(* Logix 5000 project; controller NSH_PLC1 vendor 1 type 14 code 167 rev 32.11; software revision 32.02; part 10 of 12 *)
(* tags used below, declared in another part *)
   BH3 : Motor;   // BH Rock
   CR_RunCommon : BOOL;   // PreClean, Run Common Units
   CR_StopCommon : BOOL;   // PreClean, Stop Common Units
   CR_StopLine1 : BOOL;   // Pre Clean Stop Line 1 Relay
   CR_StopPC1_FansCO : BOOL;   // Pre Clean Stop Line 1 Fans Cleanout Relay
   CR_StopPC2_FansCO : BOOL;   // Pre Clean Stop Line 2 Fans Cleanout Relay
   DummyOutput : BOOL;
   MainBin1 : MainBins;   // PreClean to Huller, Main Bin #1
   MainBin2 : MainBins;   // PreClean to Huller, Main Bin #1
   MainBin3 : MainBins;   // PreClean to Huller, Main Bin #1
   MainBin4 : MainBins;   // PreClean to Huller, Main Bin #1
   MainBin5 : MainBins;   // PreClean to Huller, Main Bin #1
   MainBin6 : MainBins;   // PreClean to Huller, Main Bin #1
   MainBin7 : MainBins;   // PreClean to Huller, Main Bin #1
   MainBin8 : MainBins;   // PreClean to Huller, Main Bin #1
   P10_5A : Motor;   // Cross Auger
   P10A : Motor;   // Elev to Bins
   P11A : Motor;   // Line1 Auger
   P11B : Motor;   // Line2 Auger
   P1A : Motor;   // DO Conv.
   P2A : Motor;   // Cross Conv.
   P3A : Motor;   // Stick Reel
   P4A : Motor;   // C. Belt
   P5A : Motor;   // Ele. to Vib
   P6A : Motor;   // Vib Splitter
   P7A : Motor;   // Screener
   P7A1 : Motor;   // Screener
   P7A2 : Motor;   // Screener
   P8A2_A : Motor;   // Destoner
   P8A2_B : Motor;   // AirLock
   P8A_A : Motor;   // Destoner
   P8A_B : Motor;   // Airlock
   P9A : Motor;   // Auger
   PBB1A : Motor;   // AirLock
   PBB2A : Motor;   // AirLock
   PD1 : Motor;   // Dirt Conv.
   PD2 : Motor;   // Incline
   PR1 : Motor;   // Rock Conv.
   PR2 : Motor;   // Inc. Rock
   PR3 : Motor;   // Belt
   PS1 : Motor;   // Stick Conv.
   PS2 : Motor;   // Inc. Stick Conv.
   PS3 : Motor;   // Twig Conv.
   PS4 : Motor;   // Twig Conv.
   TMR_LineStart1 : TIMER;   // Pre Clean Line 1 Start Warning Timer
   TMR_LineStart2 : TIMER;   // Pre Clean Line 2 Start Warning Timer
   TMR_StartPC1_FansCO : TIMER;   // Pre Clean Line 1 Fans Cleanout Start Warning Timer
   TMR_StartPC2_FansCO : TIMER;   // Pre Clean Line 2 Fans Cleanout Start Warning Timer
(* MainProgram, continued *)

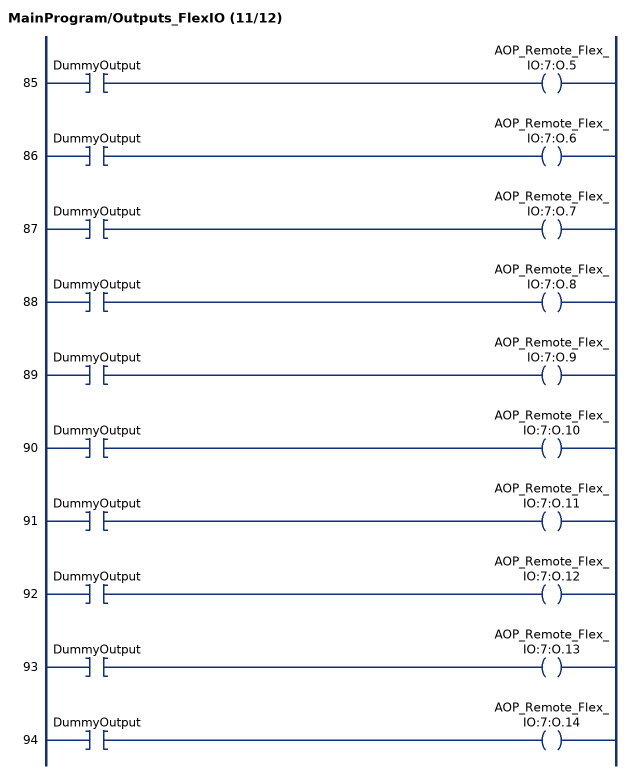
   [picture p210: MainProgram/Outputs_FlexIO rungs 85-94]
   85: XIC(DummyOutput)OTE(AOP_Remote_Flex_IO:7:O.5);
   86: XIC(DummyOutput)OTE(AOP_Remote_Flex_IO:7:O.6);
   87: XIC(DummyOutput)OTE(AOP_Remote_Flex_IO:7:O.7);
   88: XIC(DummyOutput)OTE(AOP_Remote_Flex_IO:7:O.8);
   89: XIC(DummyOutput)OTE(AOP_Remote_Flex_IO:7:O.9);
   90: XIC(DummyOutput)OTE(AOP_Remote_Flex_IO:7:O.10);
   91: XIC(DummyOutput)OTE(AOP_Remote_Flex_IO:7:O.11);
   92: XIC(DummyOutput)OTE(AOP_Remote_Flex_IO:7:O.12);
   93: XIC(DummyOutput)OTE(AOP_Remote_Flex_IO:7:O.13);
   94: XIC(DummyOutput)OTE(AOP_Remote_Flex_IO:7:O.14);
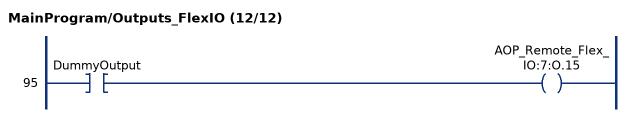
   95: XIC(DummyOutput)OTE(AOP_Remote_Flex_IO:7:O.15);
END_ROUTINE

ROUTINE Outputs_MCC1   (* ladder *)
END_ROUTINE

ROUTINE Outputs_PLC2_MCC2   (* ladder *)
END_ROUTINE

ROUTINE Outputs_PLC2_MCC3   (* ladder *)
END_ROUTINE

ROUTINE PF525_AOP_ToMotorsSUB   (* ladder *)
// Get PowerFlex525 AOP Inputs and Put Into Motor Structure
END_ROUTINE

ROUTINE PF755_AOP_ToMotorsSUB   (* ladder *)
// Get PowerFlex755 AOP Inputs and Put Into Motor Structure
END_ROUTINE
END_PROGRAM

PROGRAM PreClean   (* main routine PC_MainJSR *)
// PreClean
VAR
   CTR_HornBeeps : COUNTER := (PRE := 3);   // Number of times horn beeps
   FaultPresent : BOOL;   // A PreClean Fault is Present
   FaultReset : BOOL;   // PreClean Fault Reset
   NewFault : BOOL;   // New Precelan Fault has just occured
   NewFaultBeepHorn : BOOL;   // New Alarm, Pulse Horn
   Num_Faults : DINT;   // Number of PreCelan Faults
   Num_Faults_LS : DINT;   // Number of PreCelan Faults Last PLC Scan
   Num_Warnings : DINT;   // Number of PreCelan Warnings
   Reset_TOF_PRE : DINT;   // Reset pulse duration to Drives
   SpeedIsFactored : BOOL;   // Speed of VFD is factored by Master Speed Factor
   TempAccelerating : BOOL;   // Temp Motor is Accelerating
   TempActive : BOOL;   // Temp Motor is Active
   TempAlarm : BOOL;   // Temp Motor has Alarm
   TempAtSpeed : BOOL;   // Temp Motor is At Speed
   TempCommAlarm : BOOL;   // Temp Motor, AOP communications Alarm
   TempDecelerating : BOOL;   // Temp Motor is Decelerating
   TempFaulted : BOOL;   // Temp Motor is Faulted
   TempImbalanceTrip : BOOL;   // Temp Motor, Phase Imbalance Trip
   TempImbalanceWarning : BOOL;   // Temp Motor, Phase Imbalance Warning
   TempMainBin : MainBins := (TMR_BinFull.PRE := 20000, TMR_BinNotFull.PRE := 20000);   // Main Bin Temp
   TempMotor : Motor := (Fault_TON.PRE := 1000, Warning_TON.PRE := 1000, Reset_TOF.PRE := 500); {access None}
   TempOL_Percent : DINT;   // Temp Motor Percent Overload
   TempOverloadTrip : BOOL;   // Temp Motor, Overload Trip
   TempOverloadWarning : BOOL;   // Temp Motor, Overlaod Warning
   TempPhaseLossTrip : BOOL;   // Temp Motor, Phase Loss Trip
   TempReady : BOOL;   // Temp Motor is ready
   TempRunning : BOOL;   // Temp Motor is Running
   TempTriped : BOOL;   // Temp Motor Tripped
   TempVFD : VFD_Extra;   // Temp VFD Structure
   TempWarning : BOOL;   // Temp Motor Warning
   TMR_HornFlasher : TIMER := (PRE := 1000);   // Fault Horn Flasher timer
END_VAR

ROUTINE E300_StatusAlmWarnSUB   (* ladder *)
// Decode Status Bits and Set Warnings and Alarms For NRFV Motors with E300
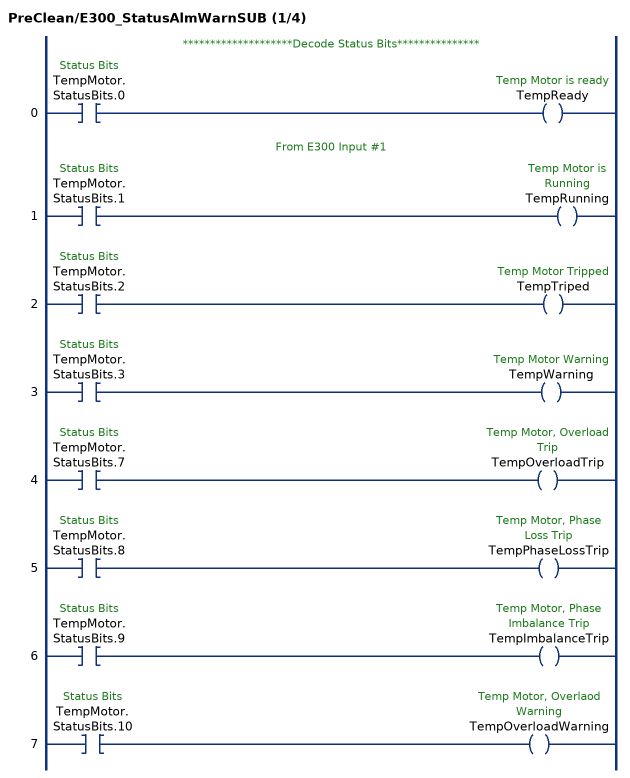
   // ********************Decode Status Bits***************
   0: XIC(TempMotor.StatusBits.0)OTE(TempReady);
   // From E300 Input #1
   1: XIC(TempMotor.StatusBits.1)OTE(TempRunning);
   2: XIC(TempMotor.StatusBits.2)OTE(TempTriped);
   3: XIC(TempMotor.StatusBits.3)OTE(TempWarning);
   4: XIC(TempMotor.StatusBits.7)OTE(TempOverloadTrip);
   5: XIC(TempMotor.StatusBits.8)OTE(TempPhaseLossTrip);
   6: XIC(TempMotor.StatusBits.9)OTE(TempImbalanceTrip);
   7: XIC(TempMotor.StatusBits.10)OTE(TempOverloadWarning);
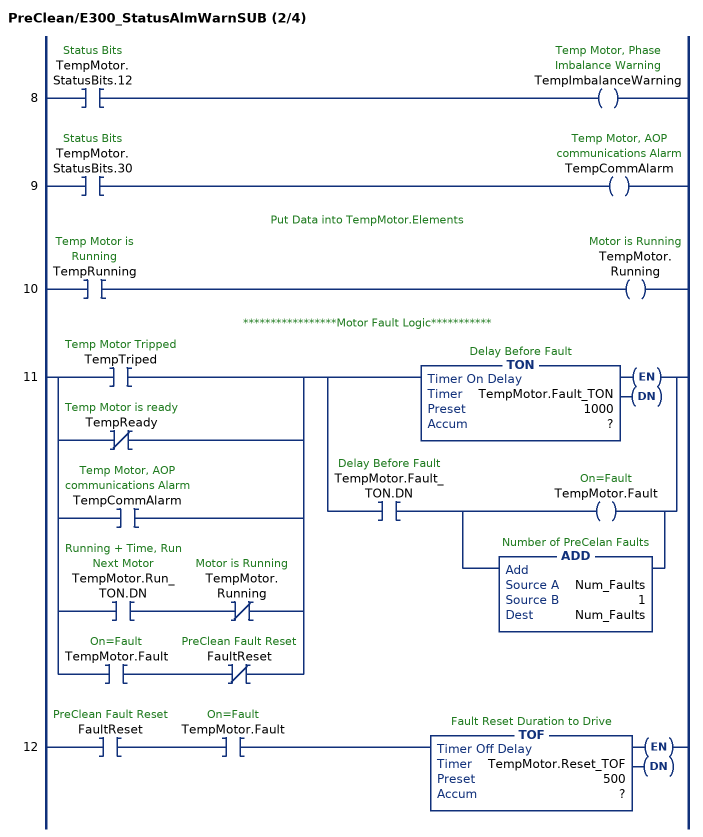
   8: XIC(TempMotor.StatusBits.12)OTE(TempImbalanceWarning);
   9: XIC(TempMotor.StatusBits.30)OTE(TempCommAlarm);
   // Put Data into TempMotor.Elements
   10: XIC(TempRunning)OTE(TempMotor.Running);
   // *****************Motor Fault Logic***********
   11: [XIC(TempTriped) ,XIO(TempReady) ,XIC(TempCommAlarm) ,XIC(TempMotor.Run_TON.DN) XIO(TempMotor.Running) ,XIC(TempMotor.Fault) XIO(FaultReset) ][TON(TempMotor.Fault_TON,?,?) ,XIC(TempMotor.Fault_TON.DN) [OTE(TempMotor.Fault) ,ADD(Num_Faults,1,Num_Faults) ] ];
   12: XIC(FaultReset)XIC(TempMotor.Fault)TOF(TempMotor.Reset_TOF,?,?);
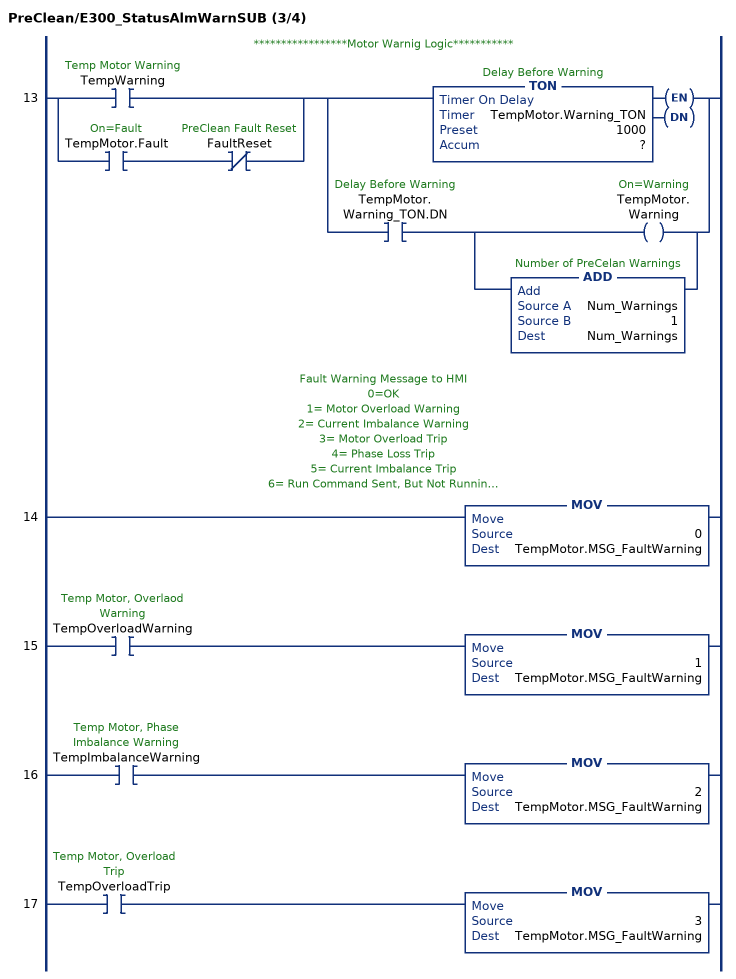
   // *****************Motor Warnig Logic***********
   13: [XIC(TempWarning) ,XIC(TempMotor.Fault) XIO(FaultReset) ][TON(TempMotor.Warning_TON,?,?) ,XIC(TempMotor.Warning_TON.DN) [OTE(TempMotor.Warning) ,ADD(Num_Warnings,1,Num_Warnings) ] ];
   // Fault Warning Message to HMI
   // 0=OK
   // 1= Motor Overload Warning
   // 2= Current Imbalance Warning
   // 3= Motor Overload Trip
   // 4= Phase Loss Trip
   // 5= Current Imbalance Trip
   // 6= Run Command Sent, But Not Running
   // 7=Loss Of Ethernet Communications
   // 8=VFD Fault
   14: MOV(0,TempMotor.MSG_FaultWarning);
   15: XIC(TempOverloadWarning)MOV(1,TempMotor.MSG_FaultWarning);
   16: XIC(TempImbalanceWarning)MOV(2,TempMotor.MSG_FaultWarning);
   17: XIC(TempOverloadTrip)MOV(3,TempMotor.MSG_FaultWarning);
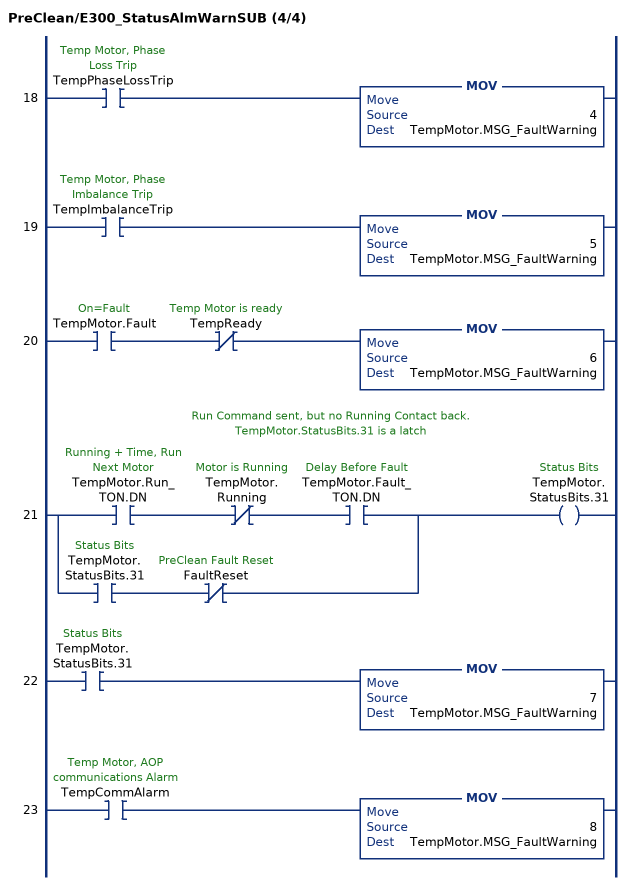
   18: XIC(TempPhaseLossTrip)MOV(4,TempMotor.MSG_FaultWarning);
   19: XIC(TempImbalanceTrip)MOV(5,TempMotor.MSG_FaultWarning);
   20: XIC(TempMotor.Fault)XIO(TempReady)MOV(6,TempMotor.MSG_FaultWarning);
   // Run Command sent, but no Running Contact back.
   // TempMotor.StatusBits.31 is a latch
   21: [XIC(TempMotor.Run_TON.DN) XIO(TempMotor.Running) XIC(TempMotor.Fault_TON.DN) ,XIC(TempMotor.StatusBits.31) XIO(FaultReset) ]OTE(TempMotor.StatusBits.31);
   22: XIC(TempMotor.StatusBits.31)MOV(7,TempMotor.MSG_FaultWarning);
   23: XIC(TempCommAlarm)MOV(8,TempMotor.MSG_FaultWarning);
END_ROUTINE

ROUTINE MainBins   (* ladder *)
// Control Main Bins
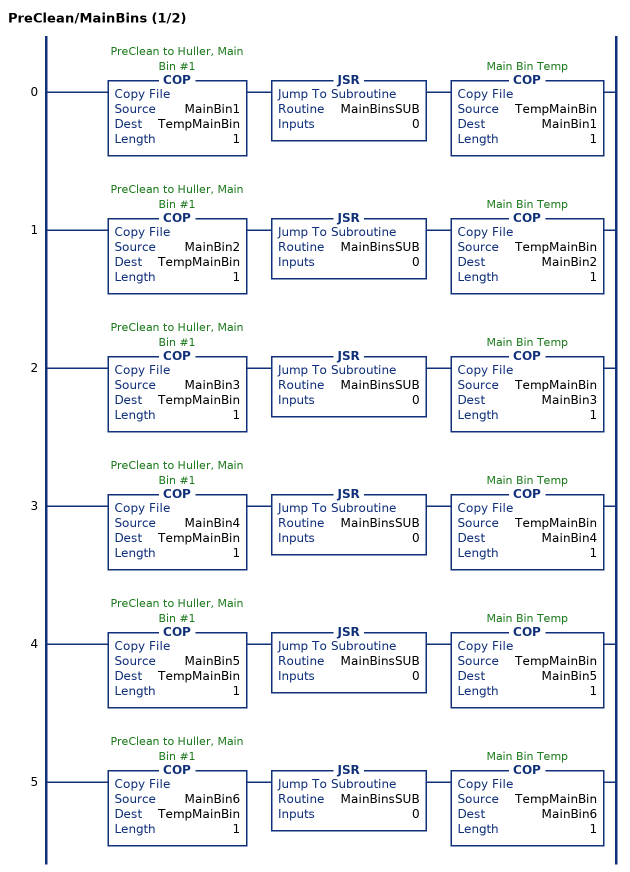
   0: COP(MainBin1,TempMainBin,1)JSR(MainBinsSUB,0)COP(TempMainBin,MainBin1,1);
   1: COP(MainBin2,TempMainBin,1)JSR(MainBinsSUB,0)COP(TempMainBin,MainBin2,1);
   2: COP(MainBin3,TempMainBin,1)JSR(MainBinsSUB,0)COP(TempMainBin,MainBin3,1);
   3: COP(MainBin4,TempMainBin,1)JSR(MainBinsSUB,0)COP(TempMainBin,MainBin4,1);
   4: COP(MainBin5,TempMainBin,1)JSR(MainBinsSUB,0)COP(TempMainBin,MainBin5,1);
   5: COP(MainBin6,TempMainBin,1)JSR(MainBinsSUB,0)COP(TempMainBin,MainBin6,1);
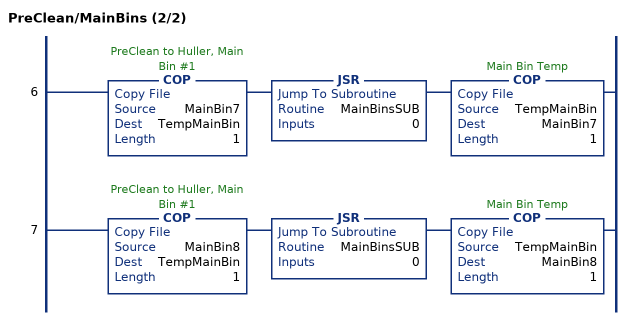
   6: COP(MainBin7,TempMainBin,1)JSR(MainBinsSUB,0)COP(TempMainBin,MainBin7,1);
   7: COP(MainBin8,TempMainBin,1)JSR(MainBinsSUB,0)COP(TempMainBin,MainBin8,1);
END_ROUTINE

ROUTINE MainBinsSUB   (* ladder *)
// Control Main Bins Switches and Lights
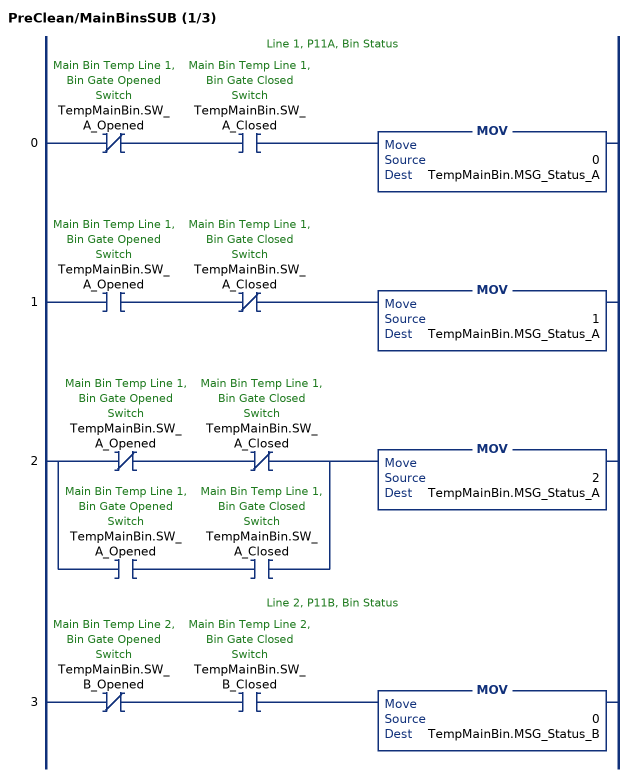
   // Line 1, P11A, Bin Status
   0: XIO(TempMainBin.SW_A_Opened)XIC(TempMainBin.SW_A_Closed)MOV(0,TempMainBin.MSG_Status_A);
   1: XIC(TempMainBin.SW_A_Opened)XIO(TempMainBin.SW_A_Closed)MOV(1,TempMainBin.MSG_Status_A);
   2: [XIO(TempMainBin.SW_A_Opened) XIO(TempMainBin.SW_A_Closed) ,XIC(TempMainBin.SW_A_Opened) XIC(TempMainBin.SW_A_Closed) ]MOV(2,TempMainBin.MSG_Status_A);
   // Line 2, P11B, Bin Status
   3: XIO(TempMainBin.SW_B_Opened)XIC(TempMainBin.SW_B_Closed)MOV(0,TempMainBin.MSG_Status_B);
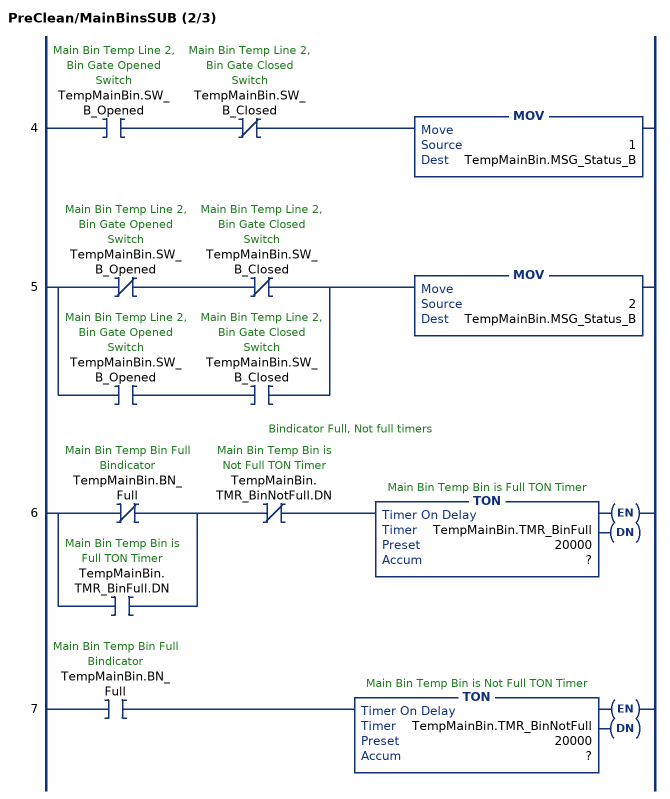
   4: XIC(TempMainBin.SW_B_Opened)XIO(TempMainBin.SW_B_Closed)MOV(1,TempMainBin.MSG_Status_B);
   5: [XIO(TempMainBin.SW_B_Opened) XIO(TempMainBin.SW_B_Closed) ,XIC(TempMainBin.SW_B_Opened) XIC(TempMainBin.SW_B_Closed) ]MOV(2,TempMainBin.MSG_Status_B);
   // Bindicator Full, Not full timers
   6: [XIO(TempMainBin.BN_Full) ,XIC(TempMainBin.TMR_BinFull.DN) ]XIO(TempMainBin.TMR_BinNotFull.DN)TON(TempMainBin.TMR_BinFull,?,?);
   7: XIC(TempMainBin.BN_Full)TON(TempMainBin.TMR_BinNotFull,?,?);
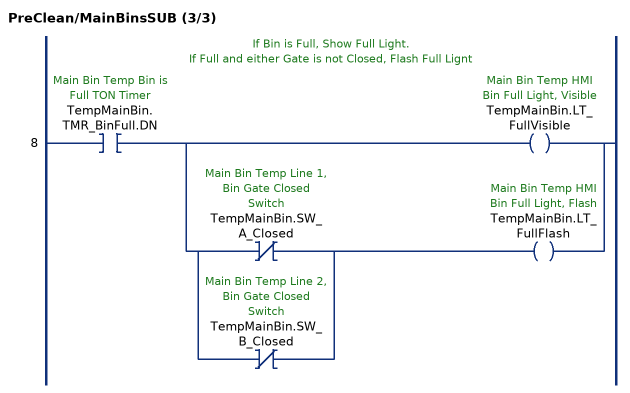
   // If Bin is Full, Show Full Light.
   // If Full and either Gate is not Closed, Flash Full Lignt
   8: XIC(TempMainBin.TMR_BinFull.DN)[OTE(TempMainBin.LT_FullVisible) ,[XIO(TempMainBin.SW_A_Closed) ,XIO(TempMainBin.SW_B_Closed) ] OTE(TempMainBin.LT_FullFlash) ];
END_ROUTINE

ROUTINE Motors   (* ladder *)
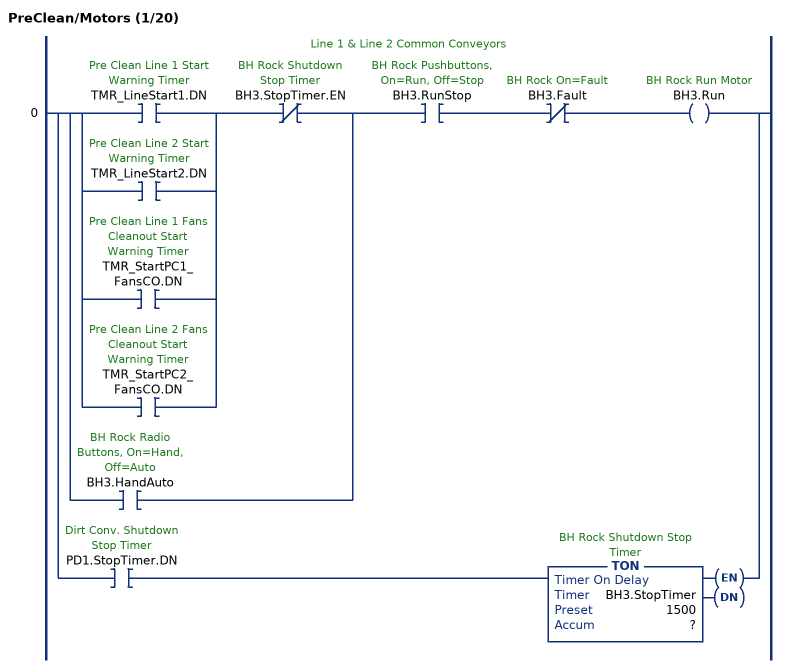
   // Line 1 & Line 2 Common Conveyors
   0: [[[XIC(TMR_LineStart1.DN) ,XIC(TMR_LineStart2.DN) ,XIC(TMR_StartPC1_FansCO.DN) ,XIC(TMR_StartPC2_FansCO.DN) ] XIO(BH3.StopTimer.EN) ,XIC(BH3.HandAuto) ] XIC(BH3.RunStop) XIO(BH3.Fault) OTE(BH3.Run) ,XIC(PD1.StopTimer.DN) TON(BH3.StopTimer,?,?) ];
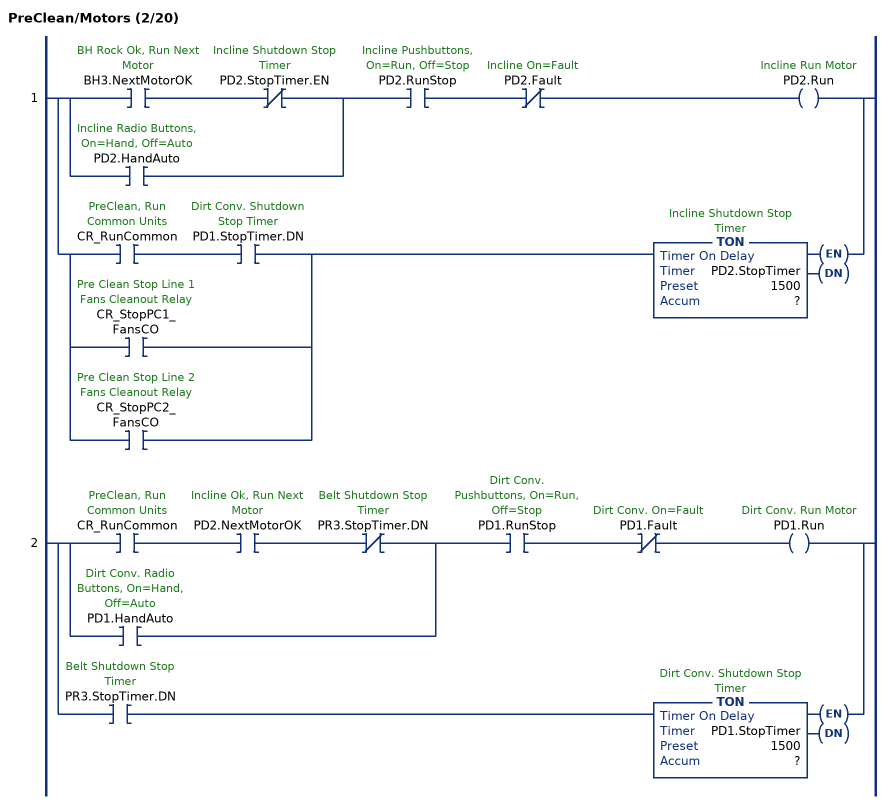
   1: [[XIC(BH3.NextMotorOK) XIO(PD2.StopTimer.EN) ,XIC(PD2.HandAuto) ] XIC(PD2.RunStop) XIO(PD2.Fault) OTE(PD2.Run) ,[XIC(CR_RunCommon) XIC(PD1.StopTimer.DN) ,XIC(CR_StopPC1_FansCO) ,XIC(CR_StopPC2_FansCO) ] TON(PD2.StopTimer,?,?) ];
   2: [[XIC(CR_RunCommon) XIC(PD2.NextMotorOK) XIO(PR3.StopTimer.DN) ,XIC(PD1.HandAuto) ] XIC(PD1.RunStop) XIO(PD1.Fault) OTE(PD1.Run) ,XIC(PR3.StopTimer.DN) TON(PD1.StopTimer,?,?) ];
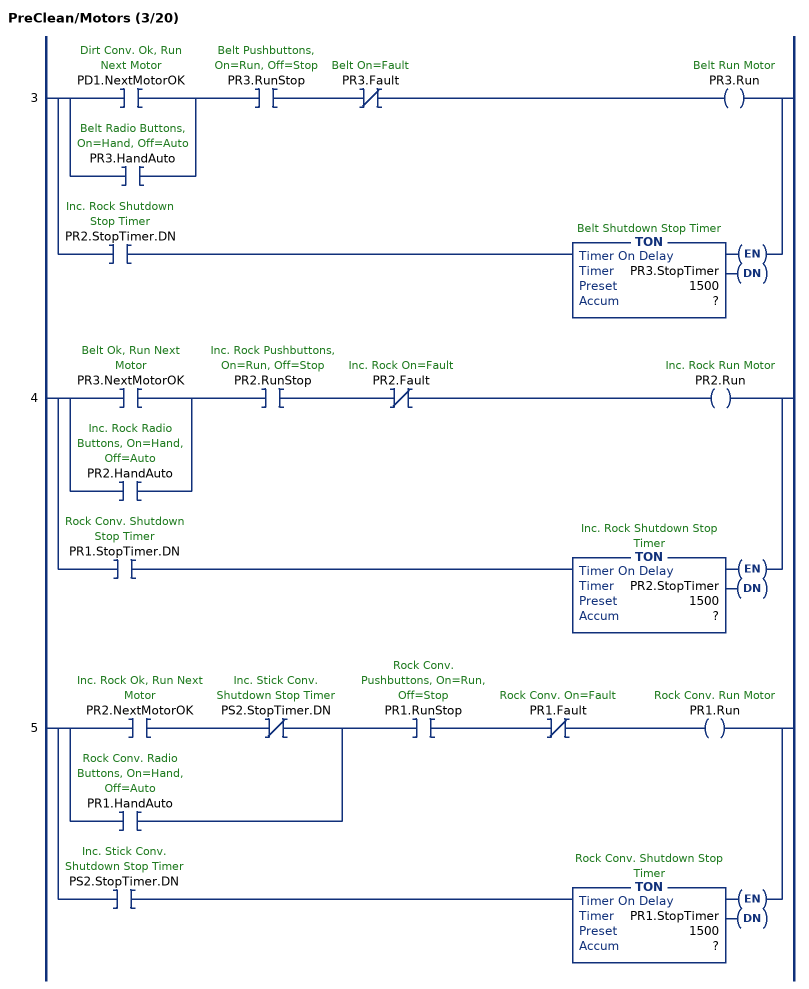
   3: [[XIC(PD1.NextMotorOK) ,XIC(PR3.HandAuto) ] XIC(PR3.RunStop) XIO(PR3.Fault) OTE(PR3.Run) ,XIC(PR2.StopTimer.DN) TON(PR3.StopTimer,?,?) ];
   4: [[XIC(PR3.NextMotorOK) ,XIC(PR2.HandAuto) ] XIC(PR2.RunStop) XIO(PR2.Fault) OTE(PR2.Run) ,XIC(PR1.StopTimer.DN) TON(PR2.StopTimer,?,?) ];
   5: [[XIC(PR2.NextMotorOK) XIO(PS2.StopTimer.DN) ,XIC(PR1.HandAuto) ] XIC(PR1.RunStop) XIO(PR1.Fault) OTE(PR1.Run) ,XIC(PS2.StopTimer.DN) TON(PR1.StopTimer,?,?) ];
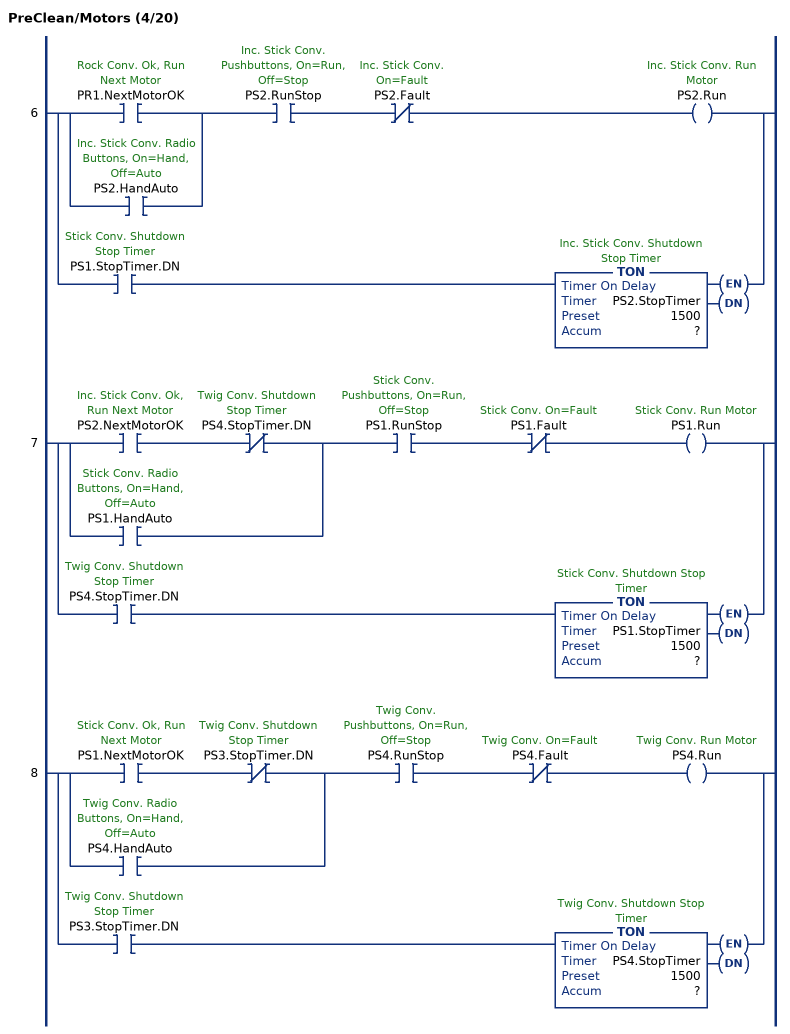
   6: [[XIC(PR1.NextMotorOK) ,XIC(PS2.HandAuto) ] XIC(PS2.RunStop) XIO(PS2.Fault) OTE(PS2.Run) ,XIC(PS1.StopTimer.DN) TON(PS2.StopTimer,?,?) ];
   7: [[XIC(PS2.NextMotorOK) XIO(PS4.StopTimer.DN) ,XIC(PS1.HandAuto) ] XIC(PS1.RunStop) XIO(PS1.Fault) OTE(PS1.Run) ,XIC(PS4.StopTimer.DN) TON(PS1.StopTimer,?,?) ];
   8: [[XIC(PS1.NextMotorOK) XIO(PS3.StopTimer.DN) ,XIC(PS4.HandAuto) ] XIC(PS4.RunStop) XIO(PS4.Fault) OTE(PS4.Run) ,XIC(PS3.StopTimer.DN) TON(PS4.StopTimer,?,?) ];
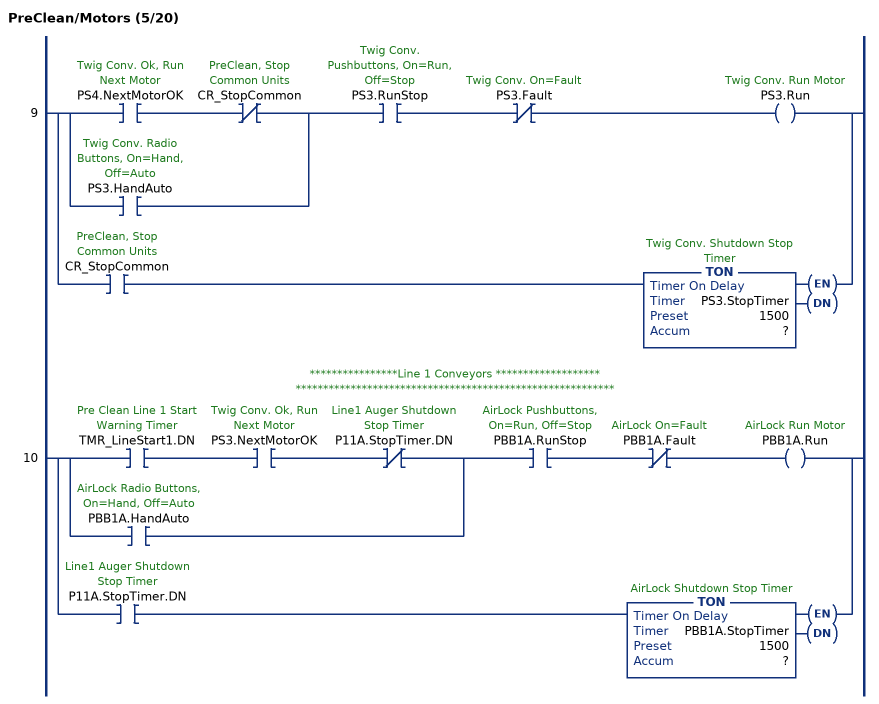
   9: [[XIC(PS4.NextMotorOK) XIO(CR_StopCommon) ,XIC(PS3.HandAuto) ] XIC(PS3.RunStop) XIO(PS3.Fault) OTE(PS3.Run) ,XIC(CR_StopCommon) TON(PS3.StopTimer,?,?) ];
   // ****************Line 1 Conveyors *******************
   //  **********************************************************
   10: [[XIC(TMR_LineStart1.DN) XIC(PS3.NextMotorOK) XIO(P11A.StopTimer.DN) ,XIC(PBB1A.HandAuto) ] XIC(PBB1A.RunStop) XIO(PBB1A.Fault) OTE(PBB1A.Run) ,XIC(P11A.StopTimer.DN) TON(PBB1A.StopTimer,?,?) ];
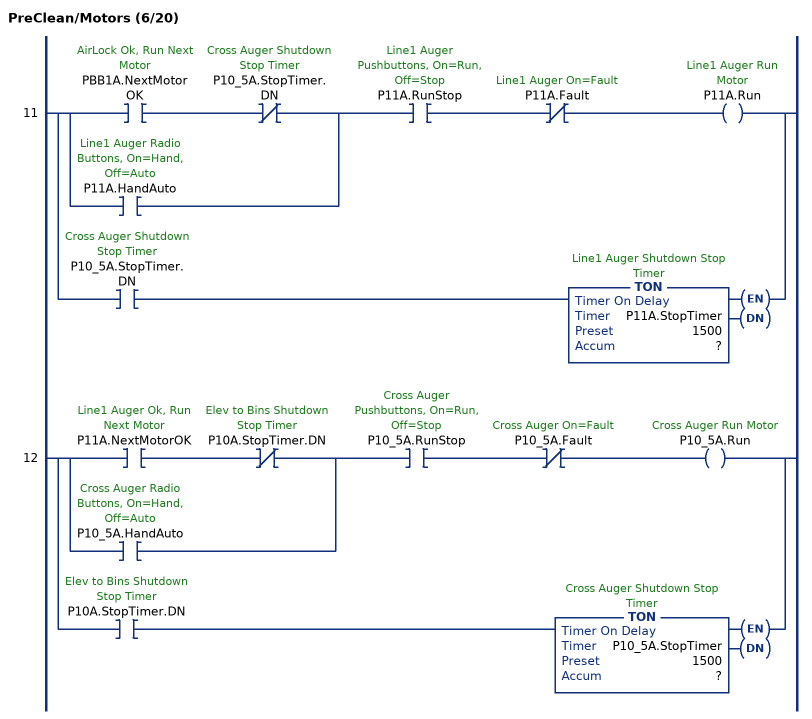
   11: [[XIC(PBB1A.NextMotorOK) XIO(P10_5A.StopTimer.DN) ,XIC(P11A.HandAuto) ] XIC(P11A.RunStop) XIO(P11A.Fault) OTE(P11A.Run) ,XIC(P10_5A.StopTimer.DN) TON(P11A.StopTimer,?,?) ];
   12: [[XIC(P11A.NextMotorOK) XIO(P10A.StopTimer.DN) ,XIC(P10_5A.HandAuto) ] XIC(P10_5A.RunStop) XIO(P10_5A.Fault) OTE(P10_5A.Run) ,XIC(P10A.StopTimer.DN) TON(P10_5A.StopTimer,?,?) ];
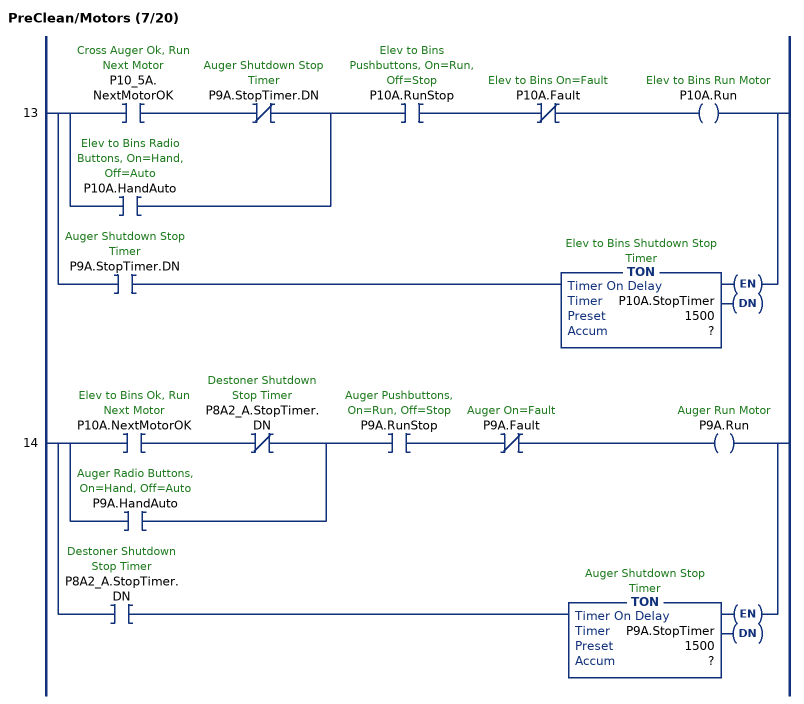
   13: [[XIC(P10_5A.NextMotorOK) XIO(P9A.StopTimer.DN) ,XIC(P10A.HandAuto) ] XIC(P10A.RunStop) XIO(P10A.Fault) OTE(P10A.Run) ,XIC(P9A.StopTimer.DN) TON(P10A.StopTimer,?,?) ];
   14: [[XIC(P10A.NextMotorOK) XIO(P8A2_A.StopTimer.DN) ,XIC(P9A.HandAuto) ] XIC(P9A.RunStop) XIO(P9A.Fault) OTE(P9A.Run) ,XIC(P8A2_A.StopTimer.DN) TON(P9A.StopTimer,?,?) ];
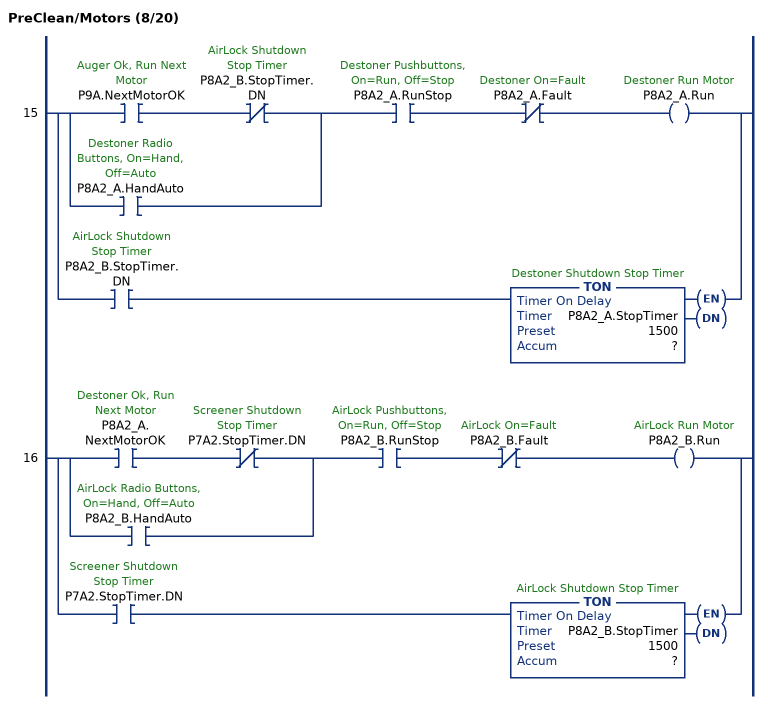
   15: [[XIC(P9A.NextMotorOK) XIO(P8A2_B.StopTimer.DN) ,XIC(P8A2_A.HandAuto) ] XIC(P8A2_A.RunStop) XIO(P8A2_A.Fault) OTE(P8A2_A.Run) ,XIC(P8A2_B.StopTimer.DN) TON(P8A2_A.StopTimer,?,?) ];
   16: [[XIC(P8A2_A.NextMotorOK) XIO(P7A2.StopTimer.DN) ,XIC(P8A2_B.HandAuto) ] XIC(P8A2_B.RunStop) XIO(P8A2_B.Fault) OTE(P8A2_B.Run) ,XIC(P7A2.StopTimer.DN) TON(P8A2_B.StopTimer,?,?) ];
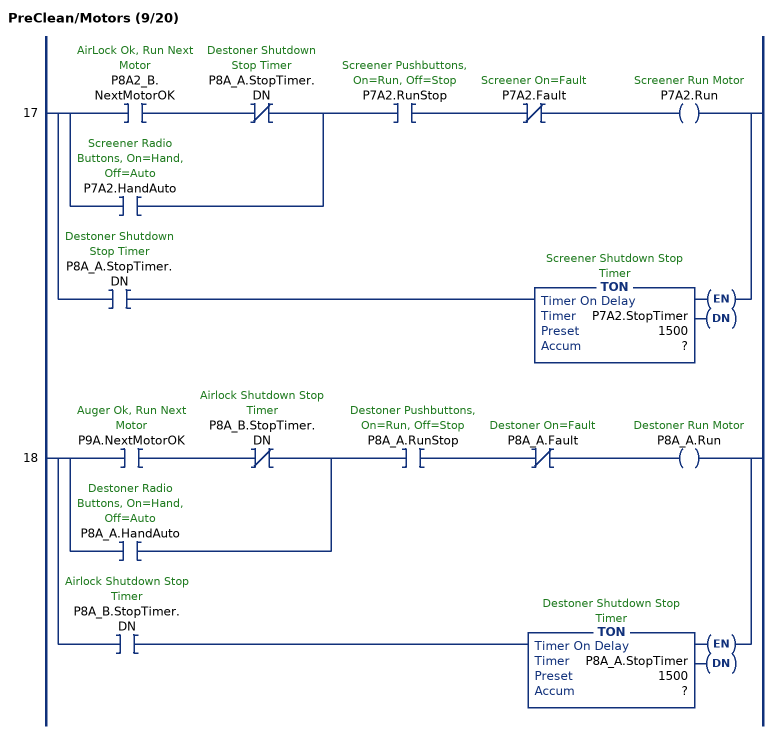
   17: [[XIC(P8A2_B.NextMotorOK) XIO(P8A_A.StopTimer.DN) ,XIC(P7A2.HandAuto) ] XIC(P7A2.RunStop) XIO(P7A2.Fault) OTE(P7A2.Run) ,XIC(P8A_A.StopTimer.DN) TON(P7A2.StopTimer,?,?) ];
   18: [[XIC(P9A.NextMotorOK) XIO(P8A_B.StopTimer.DN) ,XIC(P8A_A.HandAuto) ] XIC(P8A_A.RunStop) XIO(P8A_A.Fault) OTE(P8A_A.Run) ,XIC(P8A_B.StopTimer.DN) TON(P8A_A.StopTimer,?,?) ];
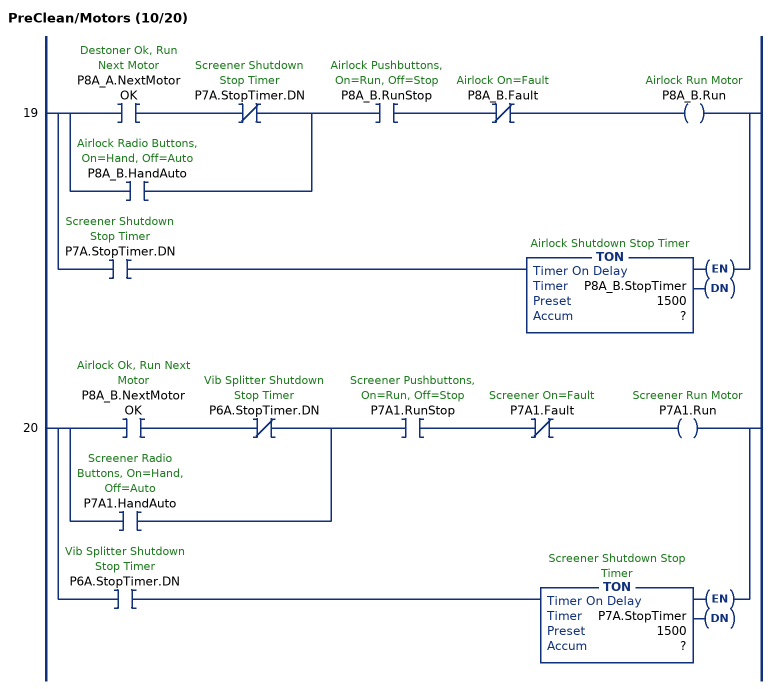
   19: [[XIC(P8A_A.NextMotorOK) XIO(P7A.StopTimer.DN) ,XIC(P8A_B.HandAuto) ] XIC(P8A_B.RunStop) XIO(P8A_B.Fault) OTE(P8A_B.Run) ,XIC(P7A.StopTimer.DN) TON(P8A_B.StopTimer,?,?) ];
   20: [[XIC(P8A_B.NextMotorOK) XIO(P6A.StopTimer.DN) ,XIC(P7A1.HandAuto) ] XIC(P7A1.RunStop) XIO(P7A1.Fault) OTE(P7A1.Run) ,XIC(P6A.StopTimer.DN) TON(P7A.StopTimer,?,?) ];
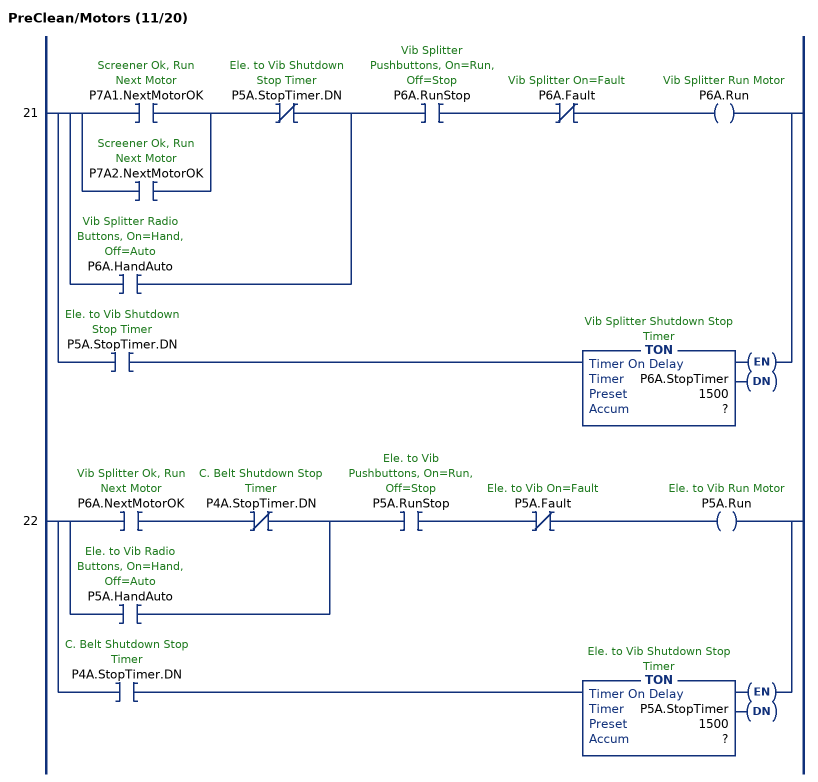
   21: [[[XIC(P7A1.NextMotorOK) ,XIC(P7A2.NextMotorOK) ] XIO(P5A.StopTimer.DN) ,XIC(P6A.HandAuto) ] XIC(P6A.RunStop) XIO(P6A.Fault) OTE(P6A.Run) ,XIC(P5A.StopTimer.DN) TON(P6A.StopTimer,?,?) ];
   22: [[XIC(P6A.NextMotorOK) XIO(P4A.StopTimer.DN) ,XIC(P5A.HandAuto) ] XIC(P5A.RunStop) XIO(P5A.Fault) OTE(P5A.Run) ,XIC(P4A.StopTimer.DN) TON(P5A.StopTimer,?,?) ];
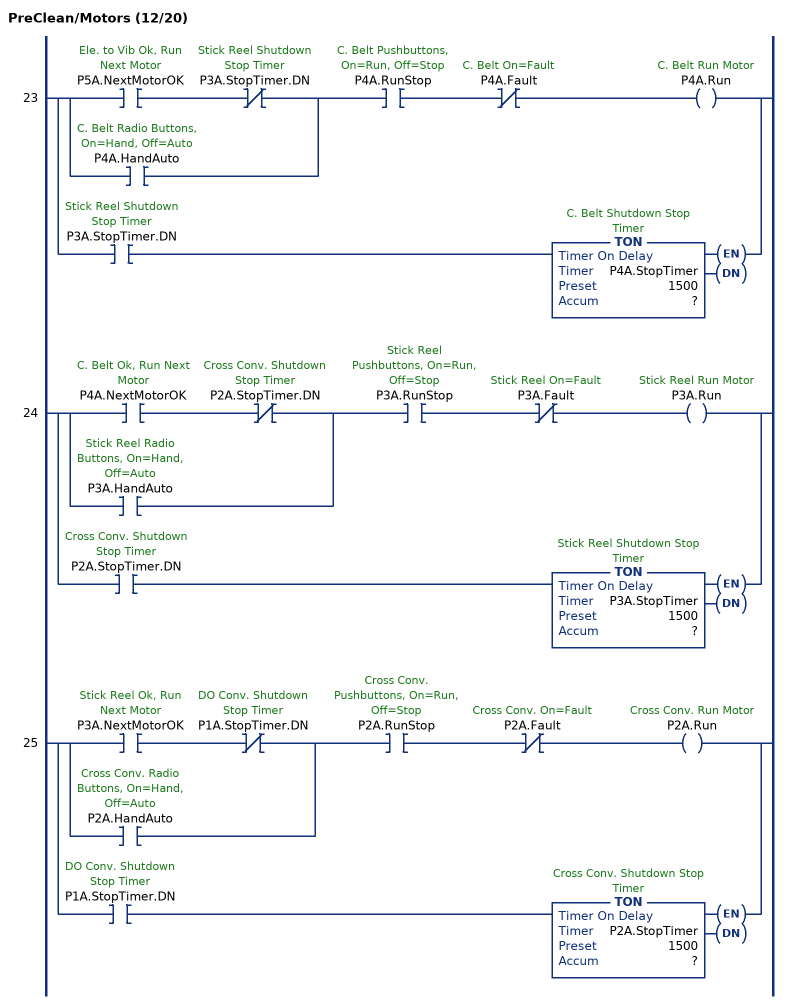
   23: [[XIC(P5A.NextMotorOK) XIO(P3A.StopTimer.DN) ,XIC(P4A.HandAuto) ] XIC(P4A.RunStop) XIO(P4A.Fault) OTE(P4A.Run) ,XIC(P3A.StopTimer.DN) TON(P4A.StopTimer,?,?) ];
   24: [[XIC(P4A.NextMotorOK) XIO(P2A.StopTimer.DN) ,XIC(P3A.HandAuto) ] XIC(P3A.RunStop) XIO(P3A.Fault) OTE(P3A.Run) ,XIC(P2A.StopTimer.DN) TON(P3A.StopTimer,?,?) ];
   25: [[XIC(P3A.NextMotorOK) XIO(P1A.StopTimer.DN) ,XIC(P2A.HandAuto) ] XIC(P2A.RunStop) XIO(P2A.Fault) OTE(P2A.Run) ,XIC(P1A.StopTimer.DN) TON(P2A.StopTimer,?,?) ];
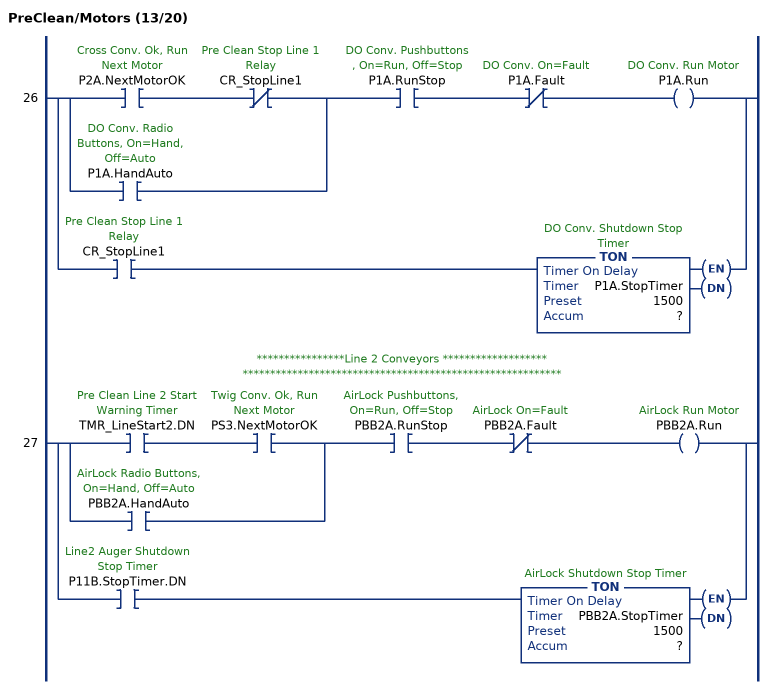
   26: [[XIC(P2A.NextMotorOK) XIO(CR_StopLine1) ,XIC(P1A.HandAuto) ] XIC(P1A.RunStop) XIO(P1A.Fault) OTE(P1A.Run) ,XIC(CR_StopLine1) TON(P1A.StopTimer,?,?) ];
   // ****************Line 2 Conveyors *******************
   //  **********************************************************
   27: [[XIC(TMR_LineStart2.DN) XIC(PS3.NextMotorOK) ,XIC(PBB2A.HandAuto) ] XIC(PBB2A.RunStop) XIO(PBB2A.Fault) OTE(PBB2A.Run) ,XIC(P11B.StopTimer.DN) TON(PBB2A.StopTimer,?,?) ];
